_CFC_ (* Continuous Function Chart, elements in execution order *)
#0 OR(SHU6_P2_UST_RE_PUSK, SHU6_P2_UST_RE_RABOTA)
#1 TON1:TON(IN: NOT #12.out 1, PT: T#500ms)
#2 RT_ModBus:R_TRIG(CLK: #1.Q)
#3 CTU_ModBus:CTU(CU: #2.Q, RESET: #3.Q, PV: 2)
#4 ADD(#3.CV, 1)
#5 WORD_TO_BYTE(#4)
#6 =(#5, 1)
#7 =(#5, 2)
#8 MUX(#5, 0, MBAddr, MBAddr_1)
#9 MUX(#5, 0, SIZEOF(RD_1), SIZEOF(RD_2))
#10 TON2:TON(IN: #1.Q, PT: T#500ms)
#11 MUX(#5, 0, ADR(RD_1), ADR(RD_2))
#12 MB_READ_REGS:ModbusRtuMaster_KL6x22B.ReadRegs(#19, Quantity, #8, #9, #11, #10.Q, T#1s)
#13 Errorld <= #12.out 3
#14 cbRead <= #12.out 4
#15 AND(#6, #12.out 2, #0)
#16 SHU6_P2_OBR_ERROR <= #15
#17 AND(#7, #12.out 2, #0)
#18 SHU6_V2_OBR_ERROR <= #17
#19 MUX(#5, 0, 2, 248)
_END_CFC_
END_PROGRAM

(* POU Persist_HVAC, CFC *)
PROGRAM Persist_HVAC
VAR
	FB_HVACPersistentDataHandling: FB_HVACPersistentDataHandling;
	_udiStatus							:	UDINT;
	_iPersistCount						:	INT;
	_bDone								:	BOOL;
	_bBusy								:	BOOL;
	_bError								:	BOOL;
	_nErrID								:	UDINT;
END_VAR
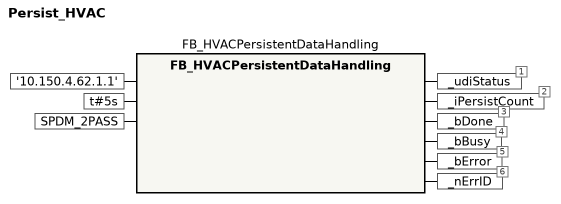
_CFC_ (* Continuous Function Chart, elements in execution order *)
#0 FB_HVACPersistentDataHandling:FB_HVACPersistentDataHandling('10.150.4.62.1.1', t#5s, SPDM_2PASS)
#1 _udiStatus <= #0.out 1
#2 _iPersistCount <= #0.out 2
#3 _bDone <= #0.out 3
#4 _bBusy <= #0.out 4
#5 _bError <= #0.out 5
#6 _nErrID <= #0.out 6
_END_CFC_
END_PROGRAM

(* POU IM/MP2/CHASTOTA_MP2_OLD, CFC *)
PROGRAM CHASTOTA_MP2_OLD
VAR
	RR: RAMP_REAL;
	SR_START_STER_REG: SR;
	SR_START_POV_REG: RS;
	RT_KOMVKL: R_TRIG;
	RT_KOMVKL_2: R_TRIG;
	RT_KOMVKL_1: R_TRIG;
	Zad_PE: TON;
END_VAR
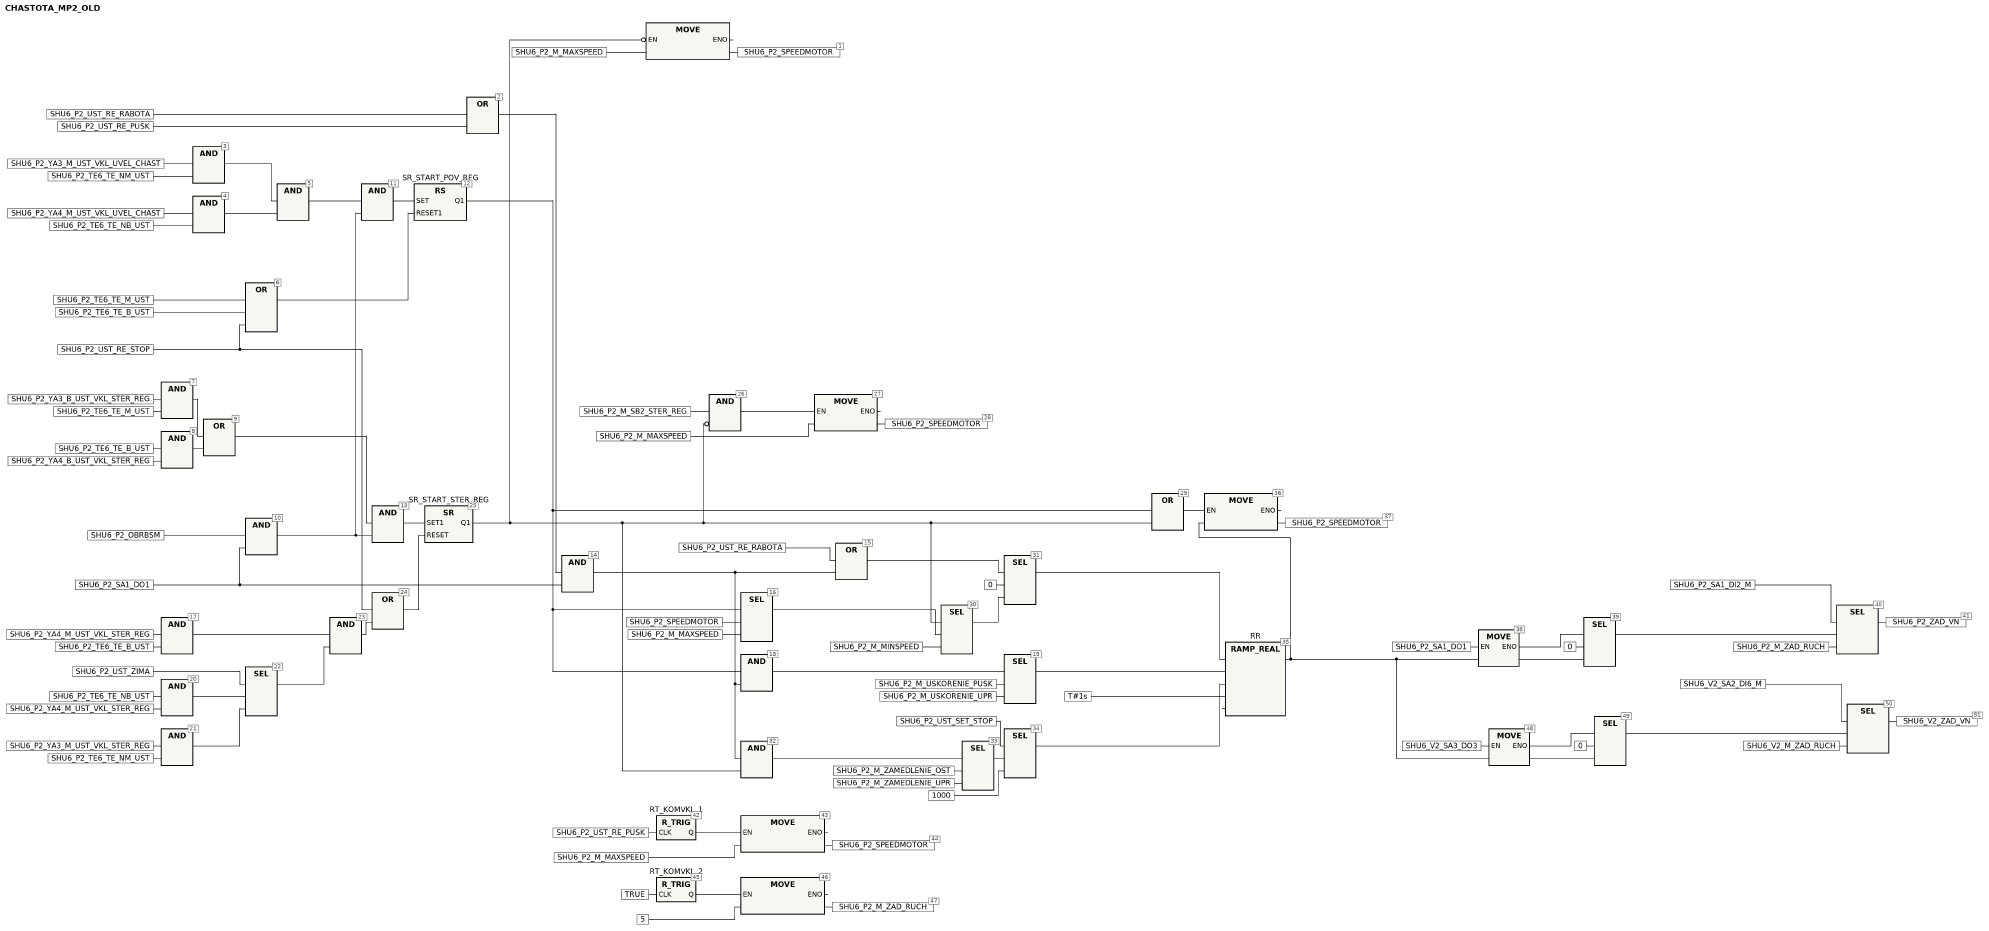
